// TIA Portal V20 export
TYPE "CMInterface_AO"
   STRUCT
      ValueOut { ExternalAccessible := 'False'; ExternalVisible := 'False'; ExternalWritable := 'False'} : Real;
   END_STRUCT;
END_TYPE
